// Mitsubishi GX Works2 project: BookEX5_5 FBcall   PLC: Q13UDV

// global labels: Global
VAR_GLOBAL
  bVar0 AT M5000 : BOOL;
  abArray0 AT M5010 : ARRAY [0..49] OF BOOL;
  sStr0 AT D5000 : STRING[199];
  sStr1 AT D5100 : STRING[199];
  sStr2 AT D5200 : STRING[199];
  sStr3 AT D5300 : STRING[199];
  sStr4 AT D5400 : STRING[199];
  sStr5 AT D5500 : STRING[199];
  sStr6 AT D5600 : STRING[199];
  sStr7 AT D5700 : STRING[199];
  sStr8 AT D5800 : STRING[199];
  sStr9 AT D5900 : STRING[199];
  iVar0 AT D4500 : INT;
  iVar1 AT D4501 : INT;
  iVar2 AT D4502 : INT;
  iVar3 AT D4503 : INT;
  iVar4 AT D4504 : INT;
  iVar5 AT D4505 : INT;
  iVar6 AT D4506 : INT;
  iVar7 AT D4507 : INT;
  iVar8 AT D4508 : INT;
  iVar9 AT D4509 : INT;
  dVar0 AT D4510 : DINT;
  dVar1 AT D4512 : DINT;
  dVar2 AT D4514 : DINT;
  dVar3 AT D4516 : DINT;
  dVar4 AT D4518 : DINT;
  dVar5 AT D4520 : DINT;
  dVar6 AT D4522 : DINT;
  dVar7 AT D4524 : DINT;
  dVar8 AT D4526 : DINT;
  dVar9 AT D4528 : DINT;
  wVar0 AT D4530 : WORD;
  wVar1 AT D4531 : WORD;
  wVar2 AT D4532 : WORD;
  wVar3 AT D4533 : WORD;
  wVar4 AT D4534 : WORD;
  wVar5 AT D4535 : WORD;
  wVar6 AT D4536 : WORD;
  wVar7 AT D4537 : WORD;
  wVar8 AT D4538 : WORD;
  wVar9 AT D4539 : WORD;
  dwVar0 AT D4540 : DWORD;
  dwVar1 AT D4542 : DWORD;
  dwVar2 AT D4544 : DWORD;
  dwVar3 AT D4546 : DWORD;
  dwVar4 AT D4548 : DWORD;
  dwVar5 AT D4550 : DWORD;
  dwVar6 AT D4552 : DWORD;
  dwVar7 AT D4554 : DWORD;
  dwVar8 AT D4556 : DWORD;
  dwVar9 AT D4558 : DWORD;
  fsVar0 AT D4560 : REAL;
  fsVar1 AT D4562 : REAL;
  fsVar2 AT D4564 : REAL;
  fsVar3 AT D4566 : REAL;
  fsVar4 AT D4568 : REAL;
  fsVar5 AT D4570 : REAL;
  fsVar6 AT D4572 : REAL;
  fsVar7 AT D4574 : REAL;
  fsVar8 AT D4576 : REAL;
  fsVar9 AT D4578 : REAL;
  fdVar0 AT D4580 : LREAL;
  tTime0 AT D4620 : TIME;
  tTime1 AT D4622 : TIME;
  tTime2 AT D4624 : TIME;
  tTime3 AT D4626 : TIME;
  tTime4 AT D4628 : TIME;
  tTime5 AT D4630 : TIME;
  tTime6 AT D4632 : TIME;
  tTime7 AT D4634 : TIME;
  tTime8 AT D4636 : TIME;
  tTime9 AT D4638 : TIME;
  tTime10 AT D4640 : TIME;
  bVar1 AT M5001 : BOOL;
  bVar2 AT M5002 : BOOL;
  bVar3 AT M5003 : BOOL;
  bVar4 AT M5004 : BOOL;
  bVar5 AT M5005 : BOOL;
  bVar6 AT M5006 : BOOL;
  bVar7 AT M5007 : BOOL;
  bVar8 AT M5008 : BOOL;
  bVar9 AT M5009 : BOOL;
  abArray1 AT M5060 : ARRAY [0..49] OF BOOL;
  abArray2 AT M5110 : ARRAY [0..49] OF BOOL;
  abArray3 AT M5160 : ARRAY [0..49] OF BOOL;
  abArray4 AT M5210 : ARRAY [0..49] OF BOOL;
  abArray5 AT M5260 : ARRAY [0..49] OF BOOL;
  abArray6 AT M5310 : ARRAY [0..49] OF BOOL;
  abArray7 AT M5360 : ARRAY [0..49] OF BOOL;
  abArray8 AT M5410 : ARRAY [0..49] OF BOOL;
  abArray9 AT M5460 : ARRAY [0..49] OF BOOL;
  fdVar1 AT D4584 : LREAL;
  fdVar2 AT D4588 : LREAL;
  fdVar3 AT D4592 : LREAL;
  fdVar4 AT D4596 : LREAL;
  fdVar5 AT D4600 : LREAL;
  fdVar6 AT D4604 : LREAL;
  fdVar7 AT D4608 : LREAL;
  fdVar8 AT D4612 : LREAL;
  fdVar9 AT D4616 : LREAL;
  aSendData AT D300 : ARRAY [0..19] OF WORD;
  aRecvData AT D100 : ARRAY [0..19] OF WORD;
  dBuffer AT D200 : ARRAY [0..19] OF WORD;
END_VAR
// user libraries (not included): HMI

PROGRAM ExWTOB
VAR
  Mov8WORD_1 : Mov8WORD;
  Mov8WORD_2 : Mov8WORD;
  newWTOB_1 : newWTOB;
  Mov8WORD_3 : Mov8WORD;
END_VAR
(* structured ladder/FBD written out as ST: instructions are called as NAME(EN, inputs, outputs); _pN, _eN, _tN stand for wires *)
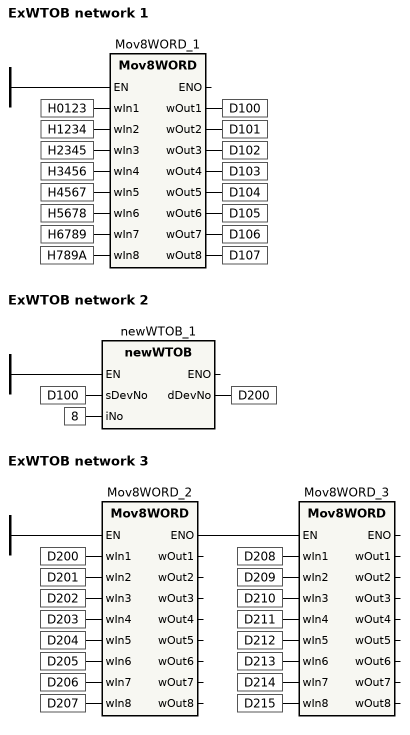
(* network 1 *)
Mov8WORD_1(EN := TRUE, wIn1 := H0123, wIn2 := H1234, wIn3 := H2345, wIn4 := H3456, wIn5 := H4567, wIn6 := H5678, wIn7 := H6789, wIn8 := H789A, wOut1 => D100, wOut2 => D101, wOut3 => D102, wOut4 => D103, wOut5 => D104, wOut6 => D105, wOut7 => D106, wOut8 => D107);
(* network 2 *)
newWTOB_1(EN := TRUE, sDevNo := D100, iNo := 8, dDevNo => D200);
(* network 3 *)
Mov8WORD_2(EN := TRUE, wIn1 := D200, wIn2 := D201, wIn3 := D202, wIn4 := D203, wIn5 := D204, wIn6 := D205, wIn7 := D206, wIn8 := D207);
Mov8WORD_3(EN := Mov8WORD_2.ENO, wIn1 := D208, wIn2 := D209, wIn3 := D210, wIn4 := D211, wIn5 := D212, wIn6 := D213, wIn7 := D214, wIn8 := D215);
END_PROGRAM

FUNCTION_BLOCK newWTOB
VAR_INPUT
  sDevNo : WORD;
  iNo : INT;
END_VAR
VAR_OUTPUT
  dDevNo : WORD;
END_VAR
VAR
  sBuffer : ARRAY [0..99] OF WORD;
  dBuffer : ARRAY [0..99] OF WORD;
  ix : INT;
END_VAR
;
BMOV(TRUE, sDevNo, iNo, sBuffer[0]); 
FOR ix := 0 TO iNo-1 DO 
		dBuffer[ix*2]  := sBuffer[ix] AND HFF;
		dBuffer[ix*2+1]:= SHR(sBuffer[ix], 8) AND HFF;
END_FOR;
BMOV(TRUE, dBuffer[0], iNo*2, dDevNo);
END_FUNCTION_BLOCK

PROGRAM ExInOut
VAR
  Mov8WORD_1 : Mov8WORD;
  Mov8WORD_2 : Mov8WORD;
  Mov8WORD_3 : Mov8WORD;
  newWTOB2_1 : newWTOB2;
  Mov8WORD_4 : Mov8WORD;
END_VAR
(* structured ladder/FBD written out as ST: instructions are called as NAME(EN, inputs, outputs); _pN, _eN, _tN stand for wires *)
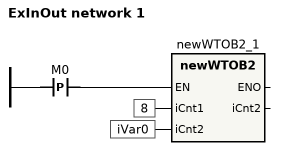
(* network 1 *)
newWTOB2_1(EN := LDP(TRUE, M0), iCnt1 := 8, iCnt2 := iVar0);
END_PROGRAM

FUNCTION_BLOCK newWTOB2
VAR_INPUT
  iCnt1 : INT;
END_VAR
VAR_IN_OUT
  iCnt2 : INT;
END_VAR
;
iCnt2 := iCnt2+iCnt1;
END_FUNCTION_BLOCK

FUNCTION_BLOCK errWTOB2
VAR_INPUT
  iCnt : INT;
END_VAR
VAR_IN_OUT
  dDevNo : ARRAY [0..19] OF WORD;
END_VAR
VAR
  wLow : WORD;
  ix : INT;
  wHigh : WORD;
END_VAR
VAR_IN_OUT
  bFlag : BOOL;
END_VAR
;
FOR ix := 0 TO iCnt-1 DO 
	wLow := dDevNo[ix] AND HFF;	
	wHigh:= SHR(dDevNo[ix], 8) AND HFF;
	dDevNo[ix+iCnt]:= wHigh;
	dDevNo[ix]  := wLow;	
END_FOR;
END_FUNCTION_BLOCK

PROGRAM ExErrInOut
VAR
  Mov8WORD_1 : Mov8WORD;
  Mov8WORD_2 : Mov8WORD;
  Mov8WORD_3 : Mov8WORD;
  Mov8WORD_4 : Mov8WORD;
  errWTOB2_1 : errWTOB2;
END_VAR
(* structured ladder/FBD written out as ST: instructions are called as NAME(EN, inputs, outputs); _pN, _eN, _tN stand for wires *)
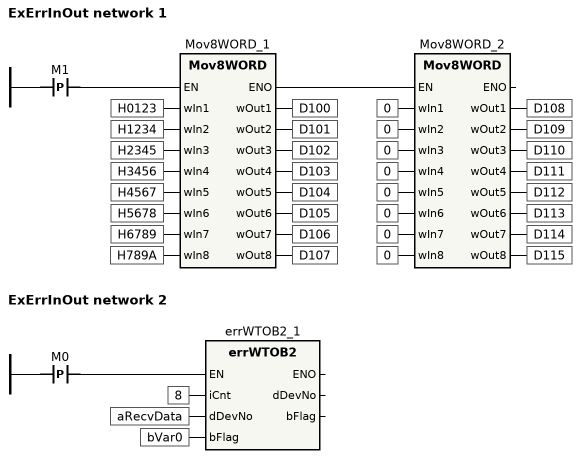
(* network 1 *)
Mov8WORD_1(EN := LDP(TRUE, M1), wIn1 := H0123, wIn2 := H1234, wIn3 := H2345, wIn4 := H3456, wIn5 := H4567, wIn6 := H5678, wIn7 := H6789, wIn8 := H789A, wOut1 => D100, wOut2 => D101, wOut3 => D102, wOut4 => D103, wOut5 => D104, wOut6 => D105, wOut7 => D106, wOut8 => D107);
Mov8WORD_2(EN := Mov8WORD_1.ENO, wIn1 := 0, wIn2 := 0, wIn3 := 0, wIn4 := 0, wIn5 := 0, wIn6 := 0, wIn7 := 0, wIn8 := 0, wOut1 => D108, wOut2 => D109, wOut3 => D110, wOut4 => D111, wOut5 => D112, wOut6 => D113, wOut7 => D114, wOut8 => D115);
(* network 2 *)
errWTOB2_1(EN := LDP(TRUE, M0), iCnt := 8, dDevNo := aRecvData, bFlag := bVar0);
END_PROGRAM
